// A dynamic collection of alarms as ST_AlarmInfo
FUNCTION_BLOCK AlarmsArray
VAR_INPUT
END_VAR
VAR_OUTPUT
END_VAR
VAR
	_malloc	: ZigaLibs_Core.FB_Malloc(0,0);
END_VAR

// Adds a new alarm defintition to the collection
METHOD AddNew
VAR_INPUT
	alarm	: ST_AlarmInfo;
END_VAR
IF NOT _malloc.IsAllocated THEN
	THIS^.Create(1);
	THIS^.GetPtr(0)^ := alarm;
ELSE
	_malloc.Expand(1);
	_malloc.Set(_malloc.Properties.NumberOfElements - 1, alarm);
END_IF
END_METHOD

// Clear the entire collection of alarms
METHOD Clear
VAR_INPUT
END_VAR
_malloc.Free();
END_METHOD

// Creates a number of alarms defined by the count value
METHOD Create : BOOL
VAR_INPUT
	count	: dint;
END_VAR
Create := _malloc.Allocate(SIZEOF(ST_AlarmInfo), count);
END_METHOD

METHOD FB_exit : BOOL
VAR_INPUT
	bInCopyCode : BOOL; // if TRUE, the exit method is called for exiting an instance that is copied afterwards (online change).
END_VAR
_malloc.Free();
END_METHOD

// Gets the pointer to the desired ST_AlarmInfo info at index
METHOD GetPtr : POINTER TO ST_AlarmInfo
VAR_INPUT
	index	: DINT;
END_VAR
GetPtr := _malloc.GetPtr(index);
END_METHOD

{attribute 'monitoring':='call'}
// Gets the total number of alarms in the collection
PROPERTY NumberOfAlarms : DINT
GET
NumberOfAlarms := _malloc.Properties.NumberOfElements;
END_GET
END_PROPERTY

// Romves an alarm at the provided index
METHOD Remove
VAR_INPUT
	index	: DINT;
END_VAR
_malloc.Remove(index);
END_METHOD

// Sets the alarm at the index to the value provided in the alarm
METHOD Set : BOOL
VAR_INPUT
	index	: DINT;
	alarm	: REFERENCE TO ST_AlarmInfo;
END_VAR
Set := _malloc.Set(index := index, value := alarm);
END_METHOD

END_FUNCTION_BLOCK

(* stored: Version 1.1.0.1
   POU AlarmsArray: Id {5ae36814-b12d-0cb1-107f-413dbe3482e3}, SpecialFunc None
   Folder Deconstructor: Id {67a941c7-1b68-0392-0007-e7b1f0861b44}
   Folder Methods - public: Id {e5146804-b4e2-0774-31c2-bc780fa2fdcb}
   Folder Properties - public: Id {87ca90bf-20ee-06e7-2e17-d480b09c82f0}
   Method AddNew: Id {2ee8993c-2570-00f1-3b4b-e879418ac64d}
   Method Clear: Id {92ed3547-8981-00da-022d-962e473da65a}
   Method Create: Id {fc4c953e-f606-0e60-282d-9b1207596240}
   Method FB_exit: Id {87506832-e9ba-0e8f-0275-a6b31064a319}
   Method GetPtr: Id {ca61ee79-678d-0197-162b-14fe24230cdb}
   Property NumberOfAlarms: Id {7d6cf9ac-d293-0789-06b6-07711939f44b}
   Get Get: Id {b4c6bcb7-e8ef-0c31-3f40-04f9718bff37}
   Method Remove: Id {0d3d4deb-38cb-044d-25d3-4040ec6dae84}
   Method Set: Id {ec4e9c2c-b666-0fb4-304e-98fde3130216} *)
